TYPE E_CoDS402HomingState :
(
	HomingInProgress,
	HomingInteruptedOrNotReached,
	HomingAttainedButNotReached,
	HomingSuccess,
	HomingError
);
END_TYPE

(* stored: Version 1.1.0.1, ProductVersion 3.1.4024.11
   DUT E_CoDS402HomingState: Id {4ed72108-9b74-459c-b2ce-f92df40503eb} *)
